(* IEC 61131-3 sources: plc_simulator/services/codesys/POUs (part 6) *)

(* ---- TSK_NoTreatment.st ---- *)
(* ===========================================================================================
 *  TSK_NoTreatment — Create no-treatment transfer tasks
 *
 *  Company : Galvatek part of the John Cockerill Group
 *  Author  : Jarmo Piipponen
 *  Created : 25.03.2026
 *
 * -------------------------------------------------------------------------------------------
 *  Scans units with a target and creates transfer tasks
 *  using the g_ntt destination table.
 *
 *  VAR_IN_OUT: io_task — only mutable array (inserts NTT tasks).
 *  All other globals are read-only via VAR_EXTERNAL.
 *
 *  ------------------------------------------------------------------------------------------
 *
 *  Changes:
 *
 *
 *
 *)

FUNCTION TSK_NoTreatment : BOOL

(* Introduction of Variables ----------------------------------------------------------------*)

VAR_INPUT
  i_time_s                  : LINT;
END_VAR

VAR_IN_OUT  (* array sizes must match GVL_JC_Constants: 3=MAX_TRANSPORTERS *)
  io_task                   : ARRAY[1..3] OF UDT_JC_TskQueueType;
END_VAR

VAR_EXTERNAL CONSTANT
    MAX_TRANSPORTERS        : INT;
    MAX_STATIONS_PER_STEP   : INT;
    MIN_STATION_INDEX        : INT;
    MAX_STATION_INDEX        : INT;
    MAX_UNITS               : INT;
    MAX_TASK_QUEUE          : INT;
    SCH_DISPATCH_MARGIN_S   : REAL;
    NOT_PROCESSED           : INT;
    PROCESSED               : INT;
    USED                    : INT;
END_VAR

VAR_EXTERNAL
  g_unit                    : ARRAY[1..MAX_UNITS] OF UDT_JC_UnitType;
  g_batch                   : ARRAY[1..MAX_UNITS] OF UDT_BatchType;
  g_ntt                     : ARRAY[1..MAX_TRANSPORTERS] OF UDT_JC_NttTransporterType;
  g_transporter             : ARRAY[1..MAX_TRANSPORTERS] OF UDT_TransporterStatusType;
  Stations                 : ARRAY[MIN_STATION_INDEX..MAX_STATION_INDEX] OF UDT_StationType;
  g_station_occupancy             : ARRAY[1..MAX_STATION_INDEX] OF UDT_JC_UnitAtStationType;
  Transporters                     : ARRAY[0..MAX_TRANSPORTERS] OF UDT_TransporterType;
  g_move                    : ARRAY[1..MAX_TRANSPORTERS] OF UDT_JC_MoveTimesType;
END_VAR

VAR
  ui                        : INT;
  loc                       : INT;
  tgt                       : INT;
  cov_t                     : INT;
  ai                        : INT;
  covers                    : BOOL;
  done                      : BOOL;
  dest                      : UDT_JC_NttDestType;
  ntt_idx                   : INT;
  on_primary                : BOOL;
  on_fallback               : BOOL;
  primary_free              : BOOL;
  dest_stn                  : INT;
  si                        : INT;
  station_idx               : INT;
  stn_free                  : BOOL;
  uj                        : INT;
  ti                        : INT;
  already                   : BOOL;
  qi2                       : INT;
  xfer_s                    : REAL;
  task_start                : LINT;
  task_end                  : LINT;
  slot_start                : LINT;
  tmp_move                  : UDT_JC_MoveTimesType;
  slot_end                  : LINT;
  latest_end                : LINT;
  travel_from_sink          : REAL;
  travel_to_lift_s          : REAL;
  trans_pos                 : INT;
  ntt_duration              : LINT;
  slot_ok                   : BOOL;
  sh                        : INT;

  (* Idle-stretch: extend blocking batch CalTime to make room for NTT -----------------------*)
  stretch_pending           : BOOL;
  stretch_unit_id           : INT;
  stretch_deficit           : DINT;
  stretch_avail             : DINT;

  (* Multi-transporter shared-area idle check -----------------------------------------------*)
  ot                        : INT;
  oq                        : INT;
  overlap_conflict          : BOOL;
  dest_x                    : DINT;
  avoid_dist                : DINT;
  cov_min_x                 : DINT;
  cov_max_x                 : DINT;
  ot_min_x                  : DINT;
  ot_max_x                  : DINT;
  zone_min_x                : DINT;
  zone_max_x                : DINT;
  danger_min                : DINT;
  danger_max                : DINT;
  (* Shared-area timing: NTT split into own-area + shared-area portions ---------------------*)
  loc_idx                   : INT;
  loc_x                     : DINT;
  phase2_s                  : REAL;
  shared_entry              : LINT;
  shared_time               : REAL;
  ot_idle_ok                : BOOL;
  ot_idle_start             : LINT;
  ot_idle_end               : LINT;
  ot_next_lift              : INT;
  ot_dispatch_from          : INT;
  ot_travel_to_next         : REAL;

  (* Idle-stretch for other transporter: widen idle gap by extending blocker CalTime --------*)
  ot_stretch_pending        : BOOL;
  ot_stretch_unit_id        : INT;
  ot_stretch_deficit        : DINT;
  ot_stretch_avail          : DINT;
  ot_stretch_need           : LINT;
  ot_stretch_ok             : BOOL;
END_VAR

TSK_NoTreatment := TRUE;

FOR ui := 1 TO MAX_UNITS DO
  tgt := g_unit[ui].Target;
  loc := g_unit[ui].location;

  IF tgt >= 1 AND tgt <= 5 AND loc >= MIN_STATION_INDEX THEN

    IF tgt = 3 AND (g_batch[ui].BatchCode = 0 OR g_batch[ui].State <> NOT_PROCESSED) THEN
      CONTINUE;
    END_IF;

    already := FALSE;
    FOR ti := 1 TO MAX_TRANSPORTERS DO
      IF NOT already THEN
        IF g_transporter[ti].Phase > 0 AND g_station_occupancy[ti].UnitId = ui THEN
          already := TRUE;
        END_IF;
        FOR qi2 := 1 TO io_task[ti].Count DO
          IF NOT already THEN
            IF io_task[ti].Queue[qi2].Unit = ui THEN
              already := TRUE;
            END_IF;
          END_IF;
        END_FOR;
      END_IF;
    END_FOR;

    IF NOT already THEN

    done := FALSE;
    FOR cov_t := 1 TO MAX_TRANSPORTERS DO
      IF NOT done THEN

      covers := FALSE;
      FOR ai := 1 TO 4 DO
        IF NOT covers THEN
          IF Transporters[cov_t].TaskArea[ai].MinLift > 0 OR Transporters[cov_t].TaskArea[ai].MaxLift > 0 THEN
            IF loc >= Transporters[cov_t].TaskArea[ai].MinLift AND loc <= Transporters[cov_t].TaskArea[ai].MaxLift THEN
              covers := TRUE;
            END_IF;
          END_IF;
        END_IF;
      END_FOR;

      IF covers AND g_transporter[cov_t].IsActive
         AND (g_transporter[cov_t].Phase = 0 OR tgt = 5) THEN

        IF tgt = 2 THEN
          IF g_batch[ui].BatchCode = 0 THEN ntt_idx := 6;
          ELSIF g_batch[ui].State = PROCESSED THEN ntt_idx := 8;
  ELSE ntt_idx := 7; END_IF;
        ELSIF tgt = 3 THEN ntt_idx := 7;
  ELSE ntt_idx := tgt; END_IF;

        dest := g_ntt[cov_t].Target[ntt_idx];

        on_primary := FALSE;
        FOR si := 1 TO dest.StationCount DO
  IF dest.Stations[si] = loc THEN on_primary := TRUE; END_IF;
        END_FOR;

        IF NOT on_primary THEN

          on_fallback := FALSE;
          FOR si := 1 TO dest.FallbackCount DO
  IF dest.FallbackStations[si] = loc THEN on_fallback := TRUE; END_IF;
          END_FOR;

          primary_free := FALSE;
          FOR si := 1 TO dest.StationCount DO
            station_idx := dest.Stations[si];
            IF station_idx <> loc AND station_idx >= MIN_STATION_INDEX AND station_idx <= MAX_STATION_INDEX THEN
              stn_free := TRUE;
              FOR uj := 1 TO MAX_UNITS DO
  IF g_unit[uj].location = station_idx AND g_unit[uj].Status = USED THEN stn_free := FALSE; END_IF;
              END_FOR;
  IF stn_free THEN primary_free := TRUE; END_IF;
            END_IF;
          END_FOR;

          dest_stn := 0;

          IF on_fallback AND NOT primary_free THEN
            dest_stn := 0;
          ELSIF on_fallback AND primary_free THEN
            FOR si := 1 TO dest.StationCount DO
              IF dest_stn = 0 THEN
                station_idx := dest.Stations[si];
                IF station_idx <> loc AND station_idx >= MIN_STATION_INDEX AND station_idx <= MAX_STATION_INDEX THEN
                  stn_free := TRUE;
                  FOR uj := 1 TO MAX_UNITS DO
  IF g_unit[uj].location = station_idx AND g_unit[uj].Status = USED THEN stn_free := FALSE; END_IF;
                  END_FOR;
  IF stn_free THEN dest_stn := station_idx; END_IF;
                END_IF;
              END_IF;
            END_FOR;
          ELSE
            FOR si := 1 TO dest.StationCount DO
              IF dest_stn = 0 THEN
                station_idx := dest.Stations[si];
                IF station_idx <> loc AND station_idx >= MIN_STATION_INDEX AND station_idx <= MAX_STATION_INDEX THEN
                  stn_free := TRUE;
                  FOR uj := 1 TO MAX_UNITS DO
  IF g_unit[uj].location = station_idx AND g_unit[uj].Status = USED THEN stn_free := FALSE; END_IF;
                  END_FOR;
  IF stn_free THEN dest_stn := station_idx; END_IF;
                END_IF;
              END_IF;
            END_FOR;

            IF dest_stn = 0 THEN
              FOR si := 1 TO dest.FallbackCount DO
                IF dest_stn = 0 THEN
                  station_idx := dest.FallbackStations[si];
                  IF station_idx <> loc AND station_idx >= MIN_STATION_INDEX AND station_idx <= MAX_STATION_INDEX THEN
                    stn_free := TRUE;
                    FOR uj := 1 TO MAX_UNITS DO
  IF g_unit[uj].location = station_idx AND g_unit[uj].Status = USED THEN stn_free := FALSE; END_IF;
                    END_FOR;
  IF stn_free THEN dest_stn := station_idx; END_IF;
                  END_IF;
                END_IF;
              END_FOR;
            END_IF;
          END_IF;

          IF dest_stn > 0 THEN
            tmp_move := g_move[cov_t];
            xfer_s := STC_CalcTransferTime(
              i_from_stn            := loc,
              i_to_stn              := dest_stn,
              i_move                := tmp_move,
              i_from_dropping_x10   := Stations[loc].DrippingTime,
              i_to_device_delay_x10 := Stations[dest_stn].DeviceDelay,
              i_drip_tray_delay_x10 := Transporters[cov_t].DripTrayDelay);

            (* ── Travel-to: time for transporter to reach lift station ── *)
            travel_to_lift_s := 0.0;
            IF g_transporter[cov_t].Phase = 0 THEN
              trans_pos := g_transporter[cov_t].CurrentStation;
            ELSE
              trans_pos := g_transporter[cov_t].SinkStationTarget;
            END_IF;
            IF trans_pos > 0 AND trans_pos <> loc THEN
              travel_to_lift_s := STC_CalcHorizontalTravel(
                i_from_stn := trans_pos,
                i_to_stn   := loc,
                i_move     := tmp_move);
            END_IF;

            task_start := i_time_s + REAL_TO_LINT(travel_to_lift_s);
            task_end   := task_start + REAL_TO_LINT(xfer_s);
            ntt_duration := task_end - task_start;

            slot_ok := FALSE;
            stretch_pending := FALSE;
            ot_stretch_pending := FALSE;

            IF io_task[cov_t].Count = 0 THEN
              slot_ok := TRUE;
            ELSE
              IF io_task[cov_t].Queue[1].StartTime > task_start THEN
                slot_start := task_start;
                slot_end   := io_task[cov_t].Queue[1].StartTime;
                travel_from_sink := STC_CalcHorizontalTravel(
                  i_from_stn := dest_stn,
                  i_to_stn   := io_task[cov_t].Queue[1].LiftStationTarget,
                  i_move     := g_move[cov_t]);
                latest_end := slot_end - REAL_TO_LINT(travel_from_sink) - 1;
                IF task_start >= slot_start AND task_end <= latest_end THEN
                  slot_ok := TRUE;
                END_IF;

                (* ── Idle-stretch: NTT slightly too long for idle window ──
                   Check if the blocking batch's treatment CalTime can be
                   extended (up to MaxTime) to widen the idle gap.  Only flag
                   the intent here; the actual g_batch write happens after
                   the multi-transporter overlap check passes. *)
                IF NOT slot_ok AND latest_end > 0 THEN
                  stretch_deficit := LINT_TO_DINT(task_end - latest_end);
                  IF stretch_deficit > 0 THEN
                    stretch_unit_id := io_task[cov_t].Queue[1].Unit;
                    IF stretch_unit_id >= 1 AND stretch_unit_id <= MAX_UNITS THEN
                      stretch_avail := g_batch[stretch_unit_id].MaxTime
                                     - g_batch[stretch_unit_id].CalTime;
                      IF stretch_avail >= stretch_deficit THEN
                        stretch_pending := TRUE;
                        slot_ok := TRUE;
                      END_IF;
                    END_IF;
                  END_IF;
                END_IF;
              END_IF;
            END_IF;

            IF NOT slot_ok THEN
              IF io_task[cov_t].Count > 0
                 AND io_task[cov_t].Queue[1].SinkStationTarget = loc THEN
                slot_ok := TRUE;
              ELSE
                dest_stn := 0;
              END_IF;
            END_IF;
          END_IF;

          (* ── Multi-transporter shared-area idle check ──
             If dest_stn is on the shared drive area between two transporters,
             the other transporter must have an idle window covering the time
             when THIS transporter is physically on the shared area.

             NTT transfer phases:
               Phase 2: lift + drip + tray  (nostin on vielä lift-asemalla)
               Phase 3: horizontal travel   (nostin liikkuu kohti dest)
               Phase 4: lower + tray + dev  (nostin on dest-asemalla)

             If lift station is NOT on shared area:
               shared_entry = task_start + phase2_s  (travel starts)
               shared_time  = xfer_s - phase2_s
             If lift station IS on shared area:
               shared_entry = task_start  (already there)
               shared_time  = xfer_s
          *)
          IF dest_stn > 0 THEN
            overlap_conflict := FALSE;
            dest_x := Stations[dest_stn].XPosition;
            avoid_dist := Transporters[cov_t].AvoidanceWidth;
            cov_min_x := Transporters[cov_t].DrivePosMin;
            cov_max_x := Transporters[cov_t].DrivePosMax;

            FOR ot := 1 TO MAX_TRANSPORTERS DO
              IF ot <> cov_t AND NOT overlap_conflict
                 AND g_transporter[ot].IsActive THEN
                ot_min_x := Transporters[ot].DrivePosMin;
                ot_max_x := Transporters[ot].DrivePosMax;

                IF cov_min_x > ot_min_x THEN zone_min_x := cov_min_x;
  ELSE zone_min_x := ot_min_x; END_IF;
                IF cov_max_x < ot_max_x THEN zone_max_x := cov_max_x;
  ELSE zone_max_x := ot_max_x; END_IF;

                IF zone_min_x >= zone_max_x THEN CONTINUE; END_IF;
                IF dest_x < zone_min_x OR dest_x > zone_max_x THEN CONTINUE; END_IF;

                danger_min := zone_min_x - avoid_dist;
                danger_max := zone_max_x + avoid_dist;

                (* ── Calculate shared-area entry time and duration ── *)
                loc_x := Stations[loc].XPosition;
                IF loc_x >= danger_min AND loc_x <= danger_max THEN
                  shared_entry := task_start;
                  shared_time  := xfer_s;
                ELSE
                  loc_idx := loc - MIN_STATION_INDEX;
                  IF loc_idx >= 1 AND loc_idx <= 25 THEN
                    phase2_s := INT_TO_REAL(g_move[cov_t].LiftTime[loc_idx]) / 10.0
                              + INT_TO_REAL(Stations[loc].DrippingTime) / 10.0
                              + INT_TO_REAL(Transporters[cov_t].DripTrayDelay) / 10.0;
                  ELSE
                    phase2_s := 0.0;
                  END_IF;
                  shared_entry := task_start + REAL_TO_LINT(phase2_s);
                  shared_time  := xfer_s - phase2_s;
  IF shared_time < 1.0 THEN shared_time := 1.0; END_IF;
                END_IF;

                (* ── Check: does other transporter have an idle window
                     that starts ≤ shared_entry and lasts ≥ shared_time? ── *)
                ot_idle_ok := FALSE;

                IF io_task[ot].Count = 0 AND g_transporter[ot].Phase = 0 THEN
                  ot_idle_ok := TRUE;
                ELSIF io_task[ot].Count = 0
                      AND g_transporter[ot].Phase >= 1
                      AND g_transporter[ot].Phase <= 4 THEN
                  (* Transporter executing task, nothing queued after.
                     Idle starts at current task finish. *)
                  ot_idle_start := g_transporter[ot].CurrentTaskFinishTime;
                  IF ot_idle_start <= shared_entry THEN
                    ot_idle_ok := TRUE;
                  END_IF;
                ELSE
                  IF io_task[ot].Count > 0 THEN
                    IF g_transporter[ot].Phase >= 1 AND g_transporter[ot].Phase <= 4 THEN
                      (* Idle gap: current task finish → next queued start *)
                      ot_idle_start := g_transporter[ot].CurrentTaskFinishTime;
                      ot_dispatch_from := g_transporter[ot].SinkStationTarget;
                    ELSE
                      ot_idle_start := task_start;
                      ot_dispatch_from := g_transporter[ot].CurrentStation;
                    END_IF;
                    ot_next_lift := io_task[ot].Queue[1].LiftStationTarget;
                    ot_travel_to_next := 0.0;
                    IF ot_dispatch_from > 0
                       AND ot_next_lift > 0
                       AND ot_dispatch_from <> ot_next_lift THEN
                      ot_travel_to_next := STC_CalcHorizontalTravel(
                        i_from_stn := ot_dispatch_from,
                        i_to_stn   := ot_next_lift,
                        i_move     := g_move[ot]);
                    END_IF;
                    ot_idle_end := io_task[ot].Queue[1].StartTime
                                 - REAL_TO_LINT(ot_travel_to_next)
                                 - REAL_TO_LINT(SCH_DISPATCH_MARGIN_S);
                    IF ot_idle_end < ot_idle_start THEN
                      ot_idle_end := ot_idle_start;
                    END_IF;
                    IF ot_idle_start <= shared_entry
                       AND ot_idle_end >= shared_entry + REAL_TO_LINT(shared_time) THEN
                      ot_idle_ok := TRUE;
                    END_IF;
                  END_IF;

                  IF NOT ot_idle_ok THEN
                    FOR oq := 1 TO io_task[ot].Count - 1 DO
                      IF NOT ot_idle_ok THEN
                        ot_idle_start := io_task[ot].Queue[oq].FinishTime;
                        ot_dispatch_from := io_task[ot].Queue[oq].SinkStationTarget;
                        ot_next_lift := io_task[ot].Queue[oq + 1].LiftStationTarget;
                        ot_travel_to_next := 0.0;
                        IF ot_dispatch_from > 0
                           AND ot_next_lift > 0
                           AND ot_dispatch_from <> ot_next_lift THEN
                          ot_travel_to_next := STC_CalcHorizontalTravel(
                            i_from_stn := ot_dispatch_from,
                            i_to_stn   := ot_next_lift,
                            i_move     := g_move[ot]);
                        END_IF;
                        ot_idle_end := io_task[ot].Queue[oq + 1].StartTime
                                     - REAL_TO_LINT(ot_travel_to_next)
                                     - REAL_TO_LINT(SCH_DISPATCH_MARGIN_S);
                        IF ot_idle_end < ot_idle_start THEN
                          ot_idle_end := ot_idle_start;
                        END_IF;
                        IF ot_idle_start <= shared_entry
                           AND ot_idle_end >= shared_entry + REAL_TO_LINT(shared_time) THEN
                          ot_idle_ok := TRUE;
                        END_IF;
                      END_IF;
                    END_FOR;
                  END_IF;

                  IF NOT ot_idle_ok AND io_task[ot].Count > 0 THEN
                    ot_idle_start := io_task[ot].Queue[io_task[ot].Count].FinishTime;
                    IF ot_idle_start <= shared_entry THEN
                      ot_idle_ok := TRUE;
                    END_IF;
                  END_IF;
                END_IF;

                IF NOT ot_idle_ok THEN
                  (* ── Idle-stretch for other transporter ──
                     Try to widen the nearest idle gap by extending the
                     blocking batch CalTime (up to MaxTime).  Only tasks
                     with Stage > 0 (regular, not NTT) are candidates. *)
                  ot_stretch_ok := FALSE;

                  (* Try gap before first task *)
                  IF io_task[ot].Count > 0
                     AND io_task[ot].Queue[1].Stage > 0 THEN
                    IF g_transporter[ot].Phase >= 1 AND g_transporter[ot].Phase <= 4 THEN
                      ot_idle_start := g_transporter[ot].CurrentTaskFinishTime;
                      ot_dispatch_from := g_transporter[ot].SinkStationTarget;
                    ELSE
                      ot_idle_start := task_start;
                      ot_dispatch_from := g_transporter[ot].CurrentStation;
                    END_IF;
                    ot_next_lift := io_task[ot].Queue[1].LiftStationTarget;
                    ot_travel_to_next := 0.0;
                    IF ot_dispatch_from > 0
                       AND ot_next_lift > 0
                       AND ot_dispatch_from <> ot_next_lift THEN
                      ot_travel_to_next := STC_CalcHorizontalTravel(
                        i_from_stn := ot_dispatch_from,
                        i_to_stn   := ot_next_lift,
                        i_move     := g_move[ot]);
                    END_IF;
                    ot_idle_end := io_task[ot].Queue[1].StartTime
                                 - REAL_TO_LINT(ot_travel_to_next)
                                 - REAL_TO_LINT(SCH_DISPATCH_MARGIN_S);
                    IF ot_idle_end < ot_idle_start THEN
                      ot_idle_end := ot_idle_start;
                    END_IF;

                    IF ot_idle_start <= shared_entry
                       AND ot_idle_end > shared_entry THEN
                      ot_stretch_need := shared_entry
                                       + REAL_TO_LINT(shared_time)
                                       - ot_idle_end;
                      IF ot_stretch_need > LINT#0 THEN
                        ot_stretch_unit_id := io_task[ot].Queue[1].Unit;
                        IF ot_stretch_unit_id >= 1
                           AND ot_stretch_unit_id <= MAX_UNITS THEN
                          ot_stretch_avail :=
                            g_batch[ot_stretch_unit_id].MaxTime
                          - g_batch[ot_stretch_unit_id].CalTime;
                          IF ot_stretch_avail >= LINT_TO_DINT(ot_stretch_need) THEN
                            ot_stretch_deficit := LINT_TO_DINT(ot_stretch_need);
                            ot_stretch_pending := TRUE;
                            ot_stretch_ok      := TRUE;
                          END_IF;
                        END_IF;
                      END_IF;
                    END_IF;
                  END_IF;

                  (* Try gaps between tasks *)
                  IF NOT ot_stretch_ok THEN
                    FOR oq := 1 TO io_task[ot].Count - 1 DO
                      IF NOT ot_stretch_ok
                         AND io_task[ot].Queue[oq + 1].Stage > 0 THEN
                        ot_idle_start := io_task[ot].Queue[oq].FinishTime;
                        ot_dispatch_from := io_task[ot].Queue[oq].SinkStationTarget;
                        ot_next_lift := io_task[ot].Queue[oq + 1].LiftStationTarget;
                        ot_travel_to_next := 0.0;
                        IF ot_dispatch_from > 0
                           AND ot_next_lift > 0
                           AND ot_dispatch_from <> ot_next_lift THEN
                          ot_travel_to_next := STC_CalcHorizontalTravel(
                            i_from_stn := ot_dispatch_from,
                            i_to_stn   := ot_next_lift,
                            i_move     := g_move[ot]);
                        END_IF;
                        ot_idle_end := io_task[ot].Queue[oq + 1].StartTime
                                     - REAL_TO_LINT(ot_travel_to_next)
                                     - REAL_TO_LINT(SCH_DISPATCH_MARGIN_S);
                        IF ot_idle_end < ot_idle_start THEN
                          ot_idle_end := ot_idle_start;
                        END_IF;

                        IF ot_idle_start <= shared_entry
                           AND ot_idle_end > shared_entry THEN
                          ot_stretch_need := shared_entry
                                           + REAL_TO_LINT(shared_time)
                                           - ot_idle_end;
                          IF ot_stretch_need > LINT#0 THEN
                            ot_stretch_unit_id := io_task[ot].Queue[oq + 1].Unit;
                            IF ot_stretch_unit_id >= 1
                               AND ot_stretch_unit_id <= MAX_UNITS THEN
                              ot_stretch_avail :=
                                g_batch[ot_stretch_unit_id].MaxTime
                              - g_batch[ot_stretch_unit_id].CalTime;
                              IF ot_stretch_avail >= LINT_TO_DINT(ot_stretch_need) THEN
                                ot_stretch_deficit := LINT_TO_DINT(ot_stretch_need);
                                ot_stretch_pending := TRUE;
                                ot_stretch_ok      := TRUE;
                              END_IF;
                            END_IF;
                          END_IF;
                        END_IF;
                      END_IF;
                    END_FOR;
                  END_IF;

                  IF ot_stretch_ok THEN
                    ot_idle_ok := TRUE;
                  ELSE
                    overlap_conflict := TRUE;
                  END_IF;
                END_IF;
              END_IF;
            END_FOR;

  IF overlap_conflict THEN dest_stn := 0; END_IF;
          END_IF;

          IF dest_stn > 0 THEN
            (* ── Commit idle-stretch: extend blocking batch CalTime ── *)
            IF stretch_pending THEN
              g_batch[stretch_unit_id].CalTime :=
                g_batch[stretch_unit_id].CalTime + stretch_deficit;
              stretch_pending := FALSE;
            END_IF;

            (* ── Commit other-transporter idle-stretch ── *)
            IF ot_stretch_pending THEN
              g_batch[ot_stretch_unit_id].CalTime :=
                g_batch[ot_stretch_unit_id].CalTime + ot_stretch_deficit;
              ot_stretch_pending := FALSE;
            END_IF;

            IF io_task[cov_t].Count < MAX_TASK_QUEUE THEN
              FOR sh := io_task[cov_t].Count TO 1 BY -1 DO
                io_task[cov_t].Queue[sh + 1] := io_task[cov_t].Queue[sh];
              END_FOR;
              io_task[cov_t].Queue[1].Unit         := ui;
              io_task[cov_t].Queue[1].Stage        := 0;
              io_task[cov_t].Queue[1].LiftStationTarget := loc;
              io_task[cov_t].Queue[1].SinkStationTarget := dest_stn;
              io_task[cov_t].Queue[1].StartTime   := task_start;
              io_task[cov_t].Queue[1].FinishTime  := task_end;
              io_task[cov_t].Queue[1].CalcTime    := 0;
              io_task[cov_t].Queue[1].MinTime     := 0;
              io_task[cov_t].Queue[1].MaxTime     := 0;
              io_task[cov_t].Queue[1].NttPrimary := 0;
              FOR si := 1 TO dest.StationCount DO
                IF dest.Stations[si] = dest_stn THEN
                  io_task[cov_t].Queue[1].NttPrimary := 1;
                END_IF;
              END_FOR;
              io_task[cov_t].Count := io_task[cov_t].Count + 1;
              done := TRUE;
            END_IF;
          END_IF;

        END_IF; (* NOT on_primary *)
      END_IF; (* covers + idle *)
      END_IF; (* NOT done *)
    END_FOR; (* transporter loop *)
    END_IF; (* NOT already *)
  END_IF; (* valid target *)
END_FOR;

END_FUNCTION

(* ---- TSK_Resolve.st ---- *)
(* ===========================================================================================
 *  TSK_Resolve — Conflict resolution
 *
 *  Company : Galvatek part of the John Cockerill Group
 *  Author  : Jarmo Piipponen
 *  Created : 25.03.2026
 *
 * -------------------------------------------------------------------------------------------
 *  Four sequential resolution phases:
 *  1. ADVANCE (chain bottleneck + suffix flex_down)
 *  2. DELAY (single-stage flex_up)
 *  3. PRECEDING_DELAY (conf stage-1)
 *  4. DELAY_PREV_PAST_NEXT (force order swap)
 *
 *  VAR_IN_OUT: io_schedule, io_task, io_batch, io_locks,
 *  io_lock_cnt — caller passes live or workspace arrays.
 *
 *  ------------------------------------------------------------------------------------------
 *
 *  Changes:
 *
 *
 *
 *)

FUNCTION TSK_Resolve : BOOL

(* Introduction of Variables ----------------------------------------------------------------*)

VAR_INPUT
  i_conf_unit               : INT;
  i_conf_stage              : INT;
  i_conf_trans              : INT;
  i_blocked_unit            : INT;
  i_blocked_stage           : INT;
  i_deficit                 : REAL;
END_VAR

VAR_IN_OUT  (* array sizes must match GVL_JC_Constants: 50=MAX_LOCKS, 10=MAX_UNITS, 3=MAX_TRANSPORTERS *)
  io_locks                  : ARRAY[1..50] OF UDT_JC_TskLockType;
  io_lock_cnt               : INT;
  io_schedule               : ARRAY[1..10] OF UDT_JC_TskScheduleType;
  io_task                   : ARRAY[1..3] OF UDT_JC_TskQueueType;
  io_batch                  : ARRAY[1..10] OF UDT_BatchType;
END_VAR

VAR_EXTERNAL CONSTANT
    MAX_TRANSPORTERS        : INT;
    MAX_UNITS               : INT;
    SCH_TSK_FLEX_FACTOR     : REAL;
END_VAR

VAR_OUTPUT
  o_solved                  : BOOL;
  o_total_delay             : REAL;
  o_total_adv               : REAL;
END_VAR

VAR
  remain                    : REAL;
  cap                       : REAL;
  amount                    : REAL;
  stage_flex                : REAL;
  is_locked_adv             : BOOL;
  is_locked_del             : BOOL;
  can_advance               : BOOL;
  can_delay                 : BOOL;
  lock_i                    : INT;
  prev_conf_stage           : INT;
  is_pcs_locked             : BOOL;
  prev_sink_stn             : INT;
  next_lift_stn             : INT;
  is_blk_adv_locked         : BOOL;
  qi                        : INT;
  chain_flex                : REAL;
  suffix_flex               : REAL;
  earlier_stg               : INT;
  earlier_flex              : REAL;
  chain_amount              : REAL;
  suffix_amount             : REAL;
  sched_blocked             : INT;
  sched_conf                : INT;
  sched_prev_conf           : INT;
  tmp_si                    : INT;
  cap_remain                : REAL;
END_VAR

TSK_Resolve := FALSE;
o_solved      := FALSE;
o_total_delay := 0.0;
o_total_adv   := 0.0;
remain        := i_deficit;

IF remain <= 0.1 THEN
  o_solved := TRUE;
  TSK_Resolve := TRUE;
  RETURN;
END_IF;

(* Lock check: blocked stage locked DELAY? cannot ADVANCE *)
is_locked_adv := FALSE;
FOR lock_i := 1 TO io_lock_cnt DO
  IF io_locks[lock_i].Unit = i_blocked_unit
     AND io_locks[lock_i].Stage = i_blocked_stage
     AND io_locks[lock_i].Direction = 2 THEN
    is_locked_adv := TRUE;
  END_IF;
END_FOR;

(* Lock check: conf stage locked ADVANCE? cannot DELAY *)
is_locked_del := FALSE;
FOR lock_i := 1 TO io_lock_cnt DO
  IF io_locks[lock_i].Unit = i_conf_unit
     AND io_locks[lock_i].Stage = i_conf_stage
     AND io_locks[lock_i].Direction = 1 THEN
    is_locked_del := TRUE;
  END_IF;
END_FOR;

can_advance := NOT is_locked_adv;
can_delay   := NOT is_locked_del;

(* Map ProgramStage to schedule array index *)
sched_blocked := 0;
IF i_blocked_unit >= 1 AND i_blocked_unit <= MAX_UNITS THEN
  FOR tmp_si := 1 TO io_schedule[i_blocked_unit].StageCount DO
    IF io_schedule[i_blocked_unit].Stages[tmp_si].ProgramStage = i_blocked_stage THEN
      sched_blocked := tmp_si; EXIT;
    END_IF;
  END_FOR;
END_IF;

sched_conf := 0;
IF i_conf_unit >= 1 AND i_conf_unit <= MAX_UNITS THEN
  FOR tmp_si := 1 TO io_schedule[i_conf_unit].StageCount DO
    IF io_schedule[i_conf_unit].Stages[tmp_si].ProgramStage = i_conf_stage THEN
      sched_conf := tmp_si; EXIT;
    END_IF;
  END_FOR;
END_IF;

(* ================================================================ *)
(* PHASE 1: ADVANCE -- advance blocked batch                       *)
(* ================================================================ *)
IF can_advance
   AND i_blocked_unit >= 1 AND i_blocked_unit <= MAX_UNITS
   AND i_blocked_stage >= 1 THEN
IF sched_blocked >= 1 AND sched_blocked <= io_schedule[i_blocked_unit].StageCount THEN

  (* Absolute flex cap: use (MaxTime - MinTime) range, not (CalcTime - MinTime).
     This prevents cumulative drift when CalcTime is adjusted across rounds. *)
  stage_flex := DINT_TO_REAL(
    io_schedule[i_blocked_unit].Stages[sched_blocked].MaxTime
    - io_schedule[i_blocked_unit].Stages[sched_blocked].MinTime);
  IF stage_flex < 0.0 THEN stage_flex := 0.0; END_IF;
  stage_flex := stage_flex * SCH_TSK_FLEX_FACTOR;
  (* Cap to actual remaining advance room *)
  cap_remain := DINT_TO_REAL(
    io_schedule[i_blocked_unit].Stages[sched_blocked].CalcTime
    - io_schedule[i_blocked_unit].Stages[sched_blocked].MinTime);
  IF cap_remain < 0.0 THEN cap_remain := 0.0; END_IF;
  IF stage_flex > cap_remain THEN stage_flex := cap_remain; END_IF;

  IF stage_flex > 0.1 THEN
    IF io_batch[i_blocked_unit].CurStage = i_blocked_stage THEN cap := 0.9;
  ELSE cap := 0.5; END_IF;

    (* Chain bottleneck search *)
    chain_flex := stage_flex;
    FOR earlier_stg := 1 TO sched_blocked - 1 DO
      earlier_flex := DINT_TO_REAL(
        io_schedule[i_blocked_unit].Stages[earlier_stg].CalcTime
        - io_schedule[i_blocked_unit].Stages[earlier_stg].MinTime);
  IF earlier_flex < 0.0 THEN earlier_flex := 0.0; END_IF;
      IF earlier_flex > 0.0 AND earlier_flex < chain_flex THEN
        chain_flex := earlier_flex;
      END_IF;
    END_FOR;

    (* CHAIN_ADVANCE *)
    chain_amount := chain_flex * cap;
  IF chain_amount > remain THEN chain_amount := remain; END_IF;

    IF chain_amount > 0.1 THEN
      io_schedule[i_blocked_unit].Stages[sched_blocked].CalcTime :=
        io_schedule[i_blocked_unit].Stages[sched_blocked].CalcTime - REAL_TO_DINT(chain_amount);
      io_schedule[i_blocked_unit].Stages[sched_blocked].ExitTime :=
        io_schedule[i_blocked_unit].Stages[sched_blocked].ExitTime - REAL_TO_LINT(chain_amount);

      STC_ShiftSchedule(i_unit := i_blocked_unit, i_from_stage := i_blocked_stage + 1,
                         i_amount := -chain_amount, io_schedule := io_schedule, io_task := io_task);

      io_batch[i_blocked_unit].CalTime :=
        io_batch[i_blocked_unit].CalTime - REAL_TO_DINT(chain_amount);
      IF io_batch[i_blocked_unit].CalTime < io_batch[i_blocked_unit].MinTime THEN
        io_batch[i_blocked_unit].CalTime := io_batch[i_blocked_unit].MinTime;
      END_IF;

      remain := remain - chain_amount;
      o_total_adv := o_total_adv + chain_amount;
    END_IF;

    (* SUFFIX_ADVANCE *)
    suffix_flex := stage_flex - chain_flex;
    IF suffix_flex > 0.1 AND remain > 0.1 THEN
      suffix_amount := suffix_flex * cap;
  IF suffix_amount > remain THEN suffix_amount := remain; END_IF;

      IF suffix_amount > 0.1 THEN
        io_schedule[i_blocked_unit].Stages[sched_blocked].CalcTime :=
          io_schedule[i_blocked_unit].Stages[sched_blocked].CalcTime - REAL_TO_DINT(suffix_amount);
        io_schedule[i_blocked_unit].Stages[sched_blocked].ExitTime :=
          io_schedule[i_blocked_unit].Stages[sched_blocked].ExitTime - REAL_TO_LINT(suffix_amount);

        STC_ShiftSchedule(i_unit := i_blocked_unit, i_from_stage := i_blocked_stage + 1,
                           i_amount := -suffix_amount, io_schedule := io_schedule, io_task := io_task);

        io_batch[i_blocked_unit].CalTime :=
          io_batch[i_blocked_unit].CalTime - REAL_TO_DINT(suffix_amount);
        IF io_batch[i_blocked_unit].CalTime < io_batch[i_blocked_unit].MinTime THEN
          io_batch[i_blocked_unit].CalTime := io_batch[i_blocked_unit].MinTime;
        END_IF;

        remain := remain - suffix_amount;
        o_total_adv := o_total_adv + suffix_amount;
      END_IF;
    END_IF;

    (* Record lock: ADVANCE on blocked stage *)
    IF io_lock_cnt < 50 THEN
      io_lock_cnt := io_lock_cnt + 1;
      io_locks[io_lock_cnt].Unit := i_blocked_unit;
      io_locks[io_lock_cnt].Stage := i_blocked_stage;
      io_locks[io_lock_cnt].Direction := 1;
    END_IF;

    IF remain <= 0.1 THEN
  o_solved := TRUE;
  TSK_Resolve := TRUE; RETURN;
    END_IF;
  END_IF;
END_IF;
END_IF;

(* ================================================================ *)
(* PHASE 2: DELAY -- delay conflict batch                          *)
(* ================================================================ *)
IF can_delay AND remain > 0.1
   AND i_conf_unit >= 1 AND i_conf_unit <= MAX_UNITS
   AND i_conf_stage >= 1 THEN
IF sched_conf >= 1 AND sched_conf <= io_schedule[i_conf_unit].StageCount THEN

  (* Absolute flex cap: use (MaxTime - MinTime) range, not (MaxTime - CalcTime).
     This prevents cumulative drift when CalcTime is adjusted across rounds. *)
  stage_flex := DINT_TO_REAL(
    io_schedule[i_conf_unit].Stages[sched_conf].MaxTime
    - io_schedule[i_conf_unit].Stages[sched_conf].MinTime);
  IF stage_flex < 0.0 THEN stage_flex := 0.0; END_IF;
  stage_flex := stage_flex * SCH_TSK_FLEX_FACTOR;
  (* Cap to actual remaining delay room *)
  cap_remain := DINT_TO_REAL(
    io_schedule[i_conf_unit].Stages[sched_conf].MaxTime
    - io_schedule[i_conf_unit].Stages[sched_conf].CalcTime);
  IF cap_remain < 0.0 THEN cap_remain := 0.0; END_IF;
  IF stage_flex > cap_remain THEN stage_flex := cap_remain; END_IF;

  IF stage_flex > 0.1 THEN
    IF io_batch[i_conf_unit].CurStage = i_conf_stage THEN cap := 0.9;
  ELSE cap := 0.5; END_IF;
    amount := stage_flex * cap;
  IF amount > remain THEN amount := remain; END_IF;

    io_schedule[i_conf_unit].Stages[sched_conf].CalcTime :=
      io_schedule[i_conf_unit].Stages[sched_conf].CalcTime + REAL_TO_DINT(amount);
    io_schedule[i_conf_unit].Stages[sched_conf].ExitTime :=
      io_schedule[i_conf_unit].Stages[sched_conf].ExitTime + REAL_TO_LINT(amount);

    STC_ShiftSchedule(i_unit := i_conf_unit, i_from_stage := i_conf_stage + 1,
                       i_amount := amount, io_schedule := io_schedule, io_task := io_task);

    IF io_batch[i_conf_unit].CurStage = i_conf_stage THEN
      io_batch[i_conf_unit].CalTime :=
        io_batch[i_conf_unit].CalTime + REAL_TO_DINT(amount);
      IF io_batch[i_conf_unit].CalTime > io_batch[i_conf_unit].MaxTime THEN
        io_batch[i_conf_unit].CalTime := io_batch[i_conf_unit].MaxTime;
      END_IF;
    END_IF;

    remain := remain - amount;
    o_total_delay := o_total_delay + amount;

    IF io_lock_cnt < 50 THEN
      io_lock_cnt := io_lock_cnt + 1;
      io_locks[io_lock_cnt].Unit := i_conf_unit;
      io_locks[io_lock_cnt].Stage := i_conf_stage;
      io_locks[io_lock_cnt].Direction := 2;
    END_IF;

    IF remain <= 0.1 THEN
  o_solved := TRUE;
  TSK_Resolve := TRUE; RETURN;
    END_IF;
  END_IF;
END_IF;
END_IF;

(* ================================================================ *)
(* PHASE 3: PRECEDING_DELAY -- delay conf batch at stage-1         *)
(* ================================================================ *)
prev_conf_stage := i_conf_stage - 1;

sched_prev_conf := 0;
IF i_conf_unit >= 1 AND i_conf_unit <= MAX_UNITS AND prev_conf_stage >= 1 THEN
  FOR tmp_si := 1 TO io_schedule[i_conf_unit].StageCount DO
    IF io_schedule[i_conf_unit].Stages[tmp_si].ProgramStage = prev_conf_stage THEN
  sched_prev_conf := tmp_si; EXIT;
    END_IF;
  END_FOR;
END_IF;

IF remain > 0.1 AND prev_conf_stage >= 1 AND i_conf_unit >= 1 AND i_conf_unit <= MAX_UNITS
   AND sched_prev_conf >= 1 THEN
  is_pcs_locked := FALSE;
  FOR lock_i := 1 TO io_lock_cnt DO
    IF io_locks[lock_i].Unit = i_conf_unit
       AND io_locks[lock_i].Stage = prev_conf_stage
       AND io_locks[lock_i].Direction = 1 THEN
      is_pcs_locked := TRUE;
    END_IF;
  END_FOR;

  IF NOT is_pcs_locked THEN
    (* Flex cap: min + factor × (max - min); available room = flex_cap - CalcTime *)
    stage_flex := DINT_TO_REAL(
      io_schedule[i_conf_unit].Stages[sched_prev_conf].MinTime
      + REAL_TO_DINT(SCH_TSK_FLEX_FACTOR * DINT_TO_REAL(
          io_schedule[i_conf_unit].Stages[sched_prev_conf].MaxTime
        - io_schedule[i_conf_unit].Stages[sched_prev_conf].MinTime))
      - io_schedule[i_conf_unit].Stages[sched_prev_conf].CalcTime);
  IF stage_flex < 0.0 THEN stage_flex := 0.0; END_IF;

    IF stage_flex > 0.1 THEN
      IF io_batch[i_conf_unit].CurStage = prev_conf_stage THEN cap := 0.9;
  ELSE cap := 0.5; END_IF;
      amount := stage_flex * cap;
  IF amount > remain THEN amount := remain; END_IF;

      io_schedule[i_conf_unit].Stages[sched_prev_conf].CalcTime :=
        io_schedule[i_conf_unit].Stages[sched_prev_conf].CalcTime + REAL_TO_DINT(amount);
      io_schedule[i_conf_unit].Stages[sched_prev_conf].ExitTime :=
        io_schedule[i_conf_unit].Stages[sched_prev_conf].ExitTime + REAL_TO_LINT(amount);
      STC_ShiftSchedule(i_unit := i_conf_unit, i_from_stage := prev_conf_stage + 1,
                         i_amount := amount, io_schedule := io_schedule, io_task := io_task);

      IF io_batch[i_conf_unit].CurStage = i_conf_stage THEN
        io_batch[i_conf_unit].CalTime :=
          io_batch[i_conf_unit].CalTime + REAL_TO_DINT(amount);
        IF io_batch[i_conf_unit].CalTime > io_batch[i_conf_unit].MaxTime THEN
          io_batch[i_conf_unit].CalTime := io_batch[i_conf_unit].MaxTime;
        END_IF;
      END_IF;

      remain := remain - amount;
      o_total_delay := o_total_delay + amount;

      IF io_lock_cnt < 50 THEN
        io_lock_cnt := io_lock_cnt + 1;
        io_locks[io_lock_cnt].Unit := i_conf_unit;
        io_locks[io_lock_cnt].Stage := prev_conf_stage;
        io_locks[io_lock_cnt].Direction := 2;
      END_IF;

      IF remain <= 0.1 THEN
  o_solved := TRUE;
  TSK_Resolve := TRUE; RETURN;
      END_IF;
    END_IF;
  END_IF;
END_IF;

(* ================================================================ *)
(* PHASE 4: DELAY_PREV_PAST_NEXT -- force order swap               *)
(* ================================================================ *)
IF remain > 0.1 AND i_blocked_unit >= 1 AND i_blocked_unit <= MAX_UNITS THEN
  prev_sink_stn := 0;
  next_lift_stn := 0;
  IF i_conf_trans >= 1 AND i_conf_trans <= MAX_TRANSPORTERS THEN
    FOR qi := 1 TO io_task[i_conf_trans].Count DO
      IF io_task[i_conf_trans].Queue[qi].Unit = i_blocked_unit
         AND io_task[i_conf_trans].Queue[qi].Stage = i_blocked_stage THEN
        prev_sink_stn := io_task[i_conf_trans].Queue[qi].SinkStationTarget;
      END_IF;
      IF io_task[i_conf_trans].Queue[qi].Unit = i_conf_unit
         AND io_task[i_conf_trans].Queue[qi].Stage = i_conf_stage THEN
        next_lift_stn := io_task[i_conf_trans].Queue[qi].LiftStationTarget;
      END_IF;
    END_FOR;
  END_IF;

  IF NOT (prev_sink_stn > 0 AND next_lift_stn > 0 AND prev_sink_stn = next_lift_stn) THEN
    is_blk_adv_locked := FALSE;
    FOR lock_i := 1 TO io_lock_cnt DO
      IF io_locks[lock_i].Unit = i_blocked_unit
         AND io_locks[lock_i].Stage = i_blocked_stage
         AND io_locks[lock_i].Direction = 1 THEN
        is_blk_adv_locked := TRUE;
      END_IF;
    END_FOR;

    IF NOT is_blk_adv_locked THEN
      (* Flex cap: min + factor × (max - min); available room = flex_cap - CalcTime *)
      stage_flex := DINT_TO_REAL(
        io_schedule[i_blocked_unit].Stages[sched_blocked].MinTime
        + REAL_TO_DINT(SCH_TSK_FLEX_FACTOR * DINT_TO_REAL(
            io_schedule[i_blocked_unit].Stages[sched_blocked].MaxTime
          - io_schedule[i_blocked_unit].Stages[sched_blocked].MinTime))
        - io_schedule[i_blocked_unit].Stages[sched_blocked].CalcTime);
  IF stage_flex < 0.0 THEN stage_flex := 0.0; END_IF;

      IF stage_flex > 0.1 THEN
        IF io_batch[i_blocked_unit].CurStage = i_blocked_stage THEN cap := 0.9;
  ELSE cap := 0.5; END_IF;
        amount := stage_flex * cap;
  IF amount > remain THEN amount := remain; END_IF;

        io_schedule[i_blocked_unit].Stages[sched_blocked].CalcTime :=
          io_schedule[i_blocked_unit].Stages[sched_blocked].CalcTime + REAL_TO_DINT(amount);
        io_schedule[i_blocked_unit].Stages[sched_blocked].ExitTime :=
          io_schedule[i_blocked_unit].Stages[sched_blocked].ExitTime + REAL_TO_LINT(amount);
        STC_ShiftSchedule(i_unit := i_blocked_unit, i_from_stage := i_blocked_stage + 1,
                           i_amount := amount, io_schedule := io_schedule, io_task := io_task);

        IF io_batch[i_blocked_unit].CurStage = i_blocked_stage THEN
          io_batch[i_blocked_unit].CalTime :=
            io_batch[i_blocked_unit].CalTime + REAL_TO_DINT(amount);
          IF io_batch[i_blocked_unit].CalTime > io_batch[i_blocked_unit].MaxTime THEN
            io_batch[i_blocked_unit].CalTime := io_batch[i_blocked_unit].MaxTime;
          END_IF;
        END_IF;

        remain := remain - amount;
        o_total_delay := o_total_delay + amount;

        IF io_lock_cnt < 50 THEN
          io_lock_cnt := io_lock_cnt + 1;
          io_locks[io_lock_cnt].Unit := i_blocked_unit;
          io_locks[io_lock_cnt].Stage := i_blocked_stage;
          io_locks[io_lock_cnt].Direction := 2;
        END_IF;

        IF remain <= 0.1 THEN
  o_solved := TRUE;
  TSK_Resolve := TRUE; RETURN;
        END_IF;
      END_IF;
    END_IF;
  END_IF;
END_IF;

END_FUNCTION

(* ---- TWA_CalcPriority.st ---- *)
(* ============================================================
   TWA_CalcPriority.st — Priority calculation for collision avoidance

   Priority rules (from transporterWorkingArea.js):
     canEvade = FALSE  → 100000 (cannot move, others must avoid)
     phase 3 (to_sink) → 200000 + (99999 - distance_to_target)
     phase 1 (to_lift) → 100000 + (99999 - distance_to_target)
     phase 0 (idle)    → 1

   Returns REAL to avoid DINT compatibility issues.
   Values fit within REAL precision (max ~300000).
   ============================================================ *)

FUNCTION TWA_CalcPriority : DINT
VAR_INPUT
  i_phase     : INT;
  i_can_evade : BOOL;
  i_x_pos     : DINT;
  i_x_target  : DINT;
END_VAR
VAR
  dist : DINT;
END_VAR

IF NOT i_can_evade THEN
  TWA_CalcPriority := DINT#100000;
  RETURN;
END_IF;

IF i_phase = 3 THEN
  dist := ABS(i_x_pos - i_x_target);
  IF dist > 99999 THEN dist := 99999; END_IF;
  TWA_CalcPriority := DINT#200000 + (DINT#99999 - dist);
ELSIF i_phase = 1 THEN
  dist := ABS(i_x_pos - i_x_target);
  IF dist > 99999 THEN dist := 99999; END_IF;
  TWA_CalcPriority := DINT#100000 + (DINT#99999 - dist);
ELSE
  TWA_CalcPriority := 1;
END_IF;

END_FUNCTION

(* ---- DEP_FB_CalcIdleSlots.st ---- *)
(* ============================================================
   DEP_FB_CalcIdleSlots — Idle slot calculation per transporter
   ============================================================
   Calculates time windows where a transporter has no tasks.
   Each gap between consecutive tasks (or before the first /
   after the last task) is an idle slot.

   Source: transporterTaskScheduler.js calculateTransporterIdleSlots()

   Expects g_task[i_trans].Queue to be already sorted by start_time
   (TSK_FB_Scheduler TASKS_SORT phase ensures this).

   Used by: DEP_FB_Scheduler (CHECK_ANALYZE phase)
   ============================================================ *)

FUNCTION_BLOCK DEP_FB_CalcIdleSlots
VAR_INPUT
  i_trans  : INT;      (* transporter index 1..3 *)
  i_time_s : LINT;     (* current simulation time (s), unix seconds *)
END_VAR
VAR_EXTERNAL CONSTANT
    MAX_Transporters   : INT;
    MAX_Units          : INT;
    DEP_MAX_IDLE_SLOTS : INT;
END_VAR

VAR_EXTERNAL
  g_task          : ARRAY[1..MAX_Transporters] OF UDT_JC_TskQueueType;
  g_dep_idle_slot : ARRAY[1..MAX_Transporters] OF UDT_JC_DepIdleSlotSetType;
  g_transporter   : ARRAY[1..MAX_Transporters] OF UDT_TransporterStatusType;
END_VAR
VAR
  qi       : INT;      (* queue index *)
  si       : INT;      (* slot index *)
  cnt      : INT;      (* task count for this transporter *)
  prev_end : LINT;     (* end time of previous task *)
  prev_sink : INT;     (* sink station of previous task *)
  gap_start : LINT;
  gap_end   : LINT;
  HORIZON  : LINT := 9999999999;   (* open-ended future — must exceed max unix timestamp *)
END_VAR

(* Guard *)
IF i_trans < 1 OR i_trans > MAX_Transporters THEN
  RETURN;
END_IF;

(* Reset output *)
g_dep_idle_slot[i_trans].Count := 0;
si := 0;
cnt := g_task[i_trans].Count;

prev_end  := i_time_s;
(* G05: Use transporter's current station as first-slot anchor *)
prev_sink := g_transporter[i_trans].CurrentStation;

FOR qi := 1 TO MAX_Units DO
  IF qi > cnt THEN
    EXIT;
  END_IF;

  gap_start := prev_end;
  gap_end   := g_task[i_trans].Queue[qi].StartTime;

  (* Only create slot if there is a meaningful gap *)
  IF gap_end > gap_start + LINT#1 THEN
    si := si + 1;
    IF si <= DEP_MAX_IDLE_SLOTS THEN
      g_dep_idle_slot[i_trans].Slots[si].StartTime   := gap_start;
      g_dep_idle_slot[i_trans].Slots[si].EndTime     := gap_end;
      g_dep_idle_slot[i_trans].Slots[si].LiftStationTarget := prev_sink;
      g_dep_idle_slot[i_trans].Slots[si].SinkStationTarget := g_task[i_trans].Queue[qi].LiftStationTarget;
    END_IF;
  END_IF;

  prev_end  := g_task[i_trans].Queue[qi].FinishTime;
  prev_sink := g_task[i_trans].Queue[qi].SinkStationTarget;
END_FOR;

(* Final slot: after last task → open-ended *)
si := si + 1;
IF si <= DEP_MAX_IDLE_SLOTS THEN
  g_dep_idle_slot[i_trans].Slots[si].StartTime   := prev_end;
  g_dep_idle_slot[i_trans].Slots[si].EndTime     := HORIZON;
  g_dep_idle_slot[i_trans].Slots[si].LiftStationTarget := prev_sink;
  g_dep_idle_slot[i_trans].Slots[si].SinkStationTarget := 0;
END_IF;

g_dep_idle_slot[i_trans].Count := si;

END_FUNCTION_BLOCK

(* ---- DEP_FB_CalcOverlap.st ---- *)
(* ============================================================
   DEP_FB_CalcOverlap — Overlap station detection
   ============================================================
   Identifies stations where multiple transporters can operate
   (task_area ranges overlap).  A station is marked as overlap
   if two or more different transporters have task_area ranges
   that cover it (either lift or sink range).

   Source: departureScheduler.js computeOverlapStations()

   Used by: DEP_FB_Scheduler (CALC phase)
   ============================================================ *)

FUNCTION_BLOCK DEP_FB_CalcOverlap
VAR_EXTERNAL CONSTANT
    MAX_Transporters    : INT;
    MIN_StationIndex : INT;
    MAX_StationIndex   : INT;
END_VAR

VAR_EXTERNAL
  g_cfg         : ARRAY[1..MAX_Transporters] OF UDT_TransporterType;
  g_dep_overlap : UDT_JC_DepOverlapType;
END_VAR
VAR
  station_idx         : INT;
  ti          : INT;
  ai          : INT;
  cover_count : INT;
  covered     : BOOL;
  area        : UDT_TaskArea;
END_VAR

g_dep_overlap.Count := 0;

(* G09: Clear full 0..200 domain first *)
FOR station_idx := 0 TO 200 DO
  g_dep_overlap.Flags[station_idx] := FALSE;
END_FOR;

FOR station_idx := MIN_StationIndex TO MAX_StationIndex DO
  cover_count := 0;

  FOR ti := 1 TO MAX_Transporters DO
    covered := FALSE;
    FOR ai := 1 TO 4 DO
      IF NOT covered THEN
        area := g_cfg[ti].TaskArea[ai];
        (* Station is covered if within lift OR sink range *)
        IF (area.MinLift > 0 AND station_idx >= area.MinLift AND station_idx <= area.MaxLift)
           OR (area.MinSink > 0 AND station_idx >= area.MinSink AND station_idx <= area.MaxSink) THEN
          covered := TRUE;
        END_IF;
      END_IF;
    END_FOR;
    IF covered THEN
      cover_count := cover_count + 1;
    END_IF;
  END_FOR;

  IF cover_count >= 2 THEN
    g_dep_overlap.Flags[station_idx] := TRUE;
    g_dep_overlap.Count := g_dep_overlap.Count + 1;
  ELSE
    g_dep_overlap.Flags[station_idx] := FALSE;
  END_IF;
END_FOR;

END_FUNCTION_BLOCK

(* ---- DEP_FB_FitTaskToSlot.st ---- *)
(* ============================================================
   DEP_FB_FitTaskToSlot — Fit a departure task into idle slots
   ============================================================
   Tries to fit a single waiting-batch task into the idle slots
   of its assigned transporter.  Calculates travel times from
   the previous task's sink to this task's lift, and from this
   task's sink to the next task's lift.

   Source: transporterTaskScheduler.js fitSingleTaskToIdleSlots()

   Flex constraint: delay cannot exceed flex_up × flexUpFactor.
   If no slot fits, o_need_extra_s reports the shortfall for
   backward chaining.

   Used by: DEP_FB_Scheduler (CHECK_ANALYZE phase)
   ============================================================ *)

FUNCTION_BLOCK DEP_FB_FitTaskToSlot
VAR_INPUT
  i_lift_stn     : INT;     (* task lift station *)
  i_sink_stn     : INT;     (* task sink station *)
  i_trans_id     : INT;     (* transporter for this task *)
  i_task_start   : LINT;    (* scheduled task start time (s), unix seconds *)
  i_task_end     : LINT;    (* scheduled task end time (s), unix seconds *)
  i_shift_s      : REAL;    (* pre-applied shift (overlap delay) *)
  i_calc_time_s  : DINT;    (* treatment calc_time (s) *)
  i_max_time_s   : DINT;    (* treatment max_time (s) *)
  i_flex_factor  : REAL;    (* flex_up usage factor, e.g. 0.5 *)
  i_margin_s     : REAL;    (* delay significance threshold (s) *)
  i_conflict_margin_s : REAL; (* slot boundary margin (s), typ. 1.0 *)
END_VAR
VAR_OUTPUT
  o_result : UDT_JC_DepFitResultType;
END_VAR
VAR_EXTERNAL CONSTANT
    MAX_Transporters   : INT;
    DEP_MAX_IDLE_SLOTS : INT;
END_VAR

VAR_EXTERNAL
  g_dep_idle_slot : ARRAY[1..MAX_Transporters] OF UDT_JC_DepIdleSlotSetType;
  g_move          : ARRAY[1..MAX_Transporters] OF UDT_JC_MoveTimesType;
END_VAR
VAR
  si          : INT;
  slot_cnt    : INT;
  slot_start  : LINT;
  slot_end    : LINT;
  from_stn    : INT;    (* previous task's sink or transporter home *)
  to_stn      : INT;    (* next task's lift *)
  travel_to   : REAL;   (* travel time: prev_sink → this lift *)
  travel_from : REAL;   (* travel time: this sink → next_lift *)
  earliest    : LINT;
  latest      : LINT;
  task_dur    : LINT;
  delay       : REAL;
  flex_up     : REAL;
  capped_flex : REAL;
  best_delay  : REAL;
  best_slot   : INT;
  found       : BOOL;
  overflow_best_delay : REAL;   (* best delay among flex-overflow slots *)
  overflow_best_slot  : INT;
  tmp_move    : UDT_JC_MoveTimesType;  (* MATIEC cannot index arrays in FUNCTION args *)
END_VAR

(* Initialize output *)
o_result.Fits         := FALSE;
o_result.DelayTime      := 0;
o_result.NeedExtraTime := 0;
o_result.TaskEndTime   := 0;
o_result.SlotIdx     := 0;
o_result.TransporterId     := i_trans_id;

IF i_trans_id < 1 OR i_trans_id > MAX_Transporters THEN
  RETURN;
END_IF;

task_dur   := i_task_end - i_task_start;
flex_up    := DINT_TO_REAL(i_max_time_s - i_calc_time_s);
IF flex_up < 0.0 THEN flex_up := 0.0; END_IF;
capped_flex := flex_up * i_flex_factor;

slot_cnt   := g_dep_idle_slot[i_trans_id].Count;
best_delay := 1.0E9;
best_slot  := 0;
found      := FALSE;
overflow_best_delay := 1.0E9;
overflow_best_slot  := 0;

tmp_move := g_move[i_trans_id];
FOR si := 1 TO DEP_MAX_IDLE_SLOTS DO
  IF si > slot_cnt THEN
    EXIT;
  END_IF;

  slot_start := g_dep_idle_slot[i_trans_id].Slots[si].StartTime;
  slot_end   := g_dep_idle_slot[i_trans_id].Slots[si].EndTime;

  (* ── Travel time: prev task sink → this lift ── *)
  from_stn := g_dep_idle_slot[i_trans_id].Slots[si].LiftStationTarget;
  travel_to := 0.0;
  IF from_stn > 0 AND from_stn <> i_lift_stn THEN
    travel_to := STC_CalcHorizontalTravel(i_from_stn := from_stn, i_to_stn := i_lift_stn, i_move := tmp_move);
  END_IF;

  (* ── Travel time: this sink → next task lift ── *)
  to_stn := g_dep_idle_slot[i_trans_id].Slots[si].SinkStationTarget;
  travel_from := 0.0;
  IF to_stn > 0 AND to_stn <> i_sink_stn THEN
    travel_from := STC_CalcHorizontalTravel(i_from_stn := i_sink_stn, i_to_stn := to_stn, i_move := tmp_move);
  END_IF;

  (* Earliest start = max(slot_start, task_start + shift) + travel_to + conflict_margin *)
  IF slot_start > (i_task_start + REAL_TO_LINT(i_shift_s)) THEN
    earliest := slot_start + REAL_TO_LINT(travel_to + i_conflict_margin_s);
  ELSE
    earliest := i_task_start + REAL_TO_LINT(i_shift_s + travel_to + i_conflict_margin_s);
  END_IF;

  (* Latest end = slot_end - travel_from - conflict_margin *)
  IF slot_end > LINT#9000000000 THEN
    (* Open-ended slot *)
    latest := LINT#9000000000;
  ELSE
    latest := slot_end - REAL_TO_LINT(travel_from + i_conflict_margin_s);
  END_IF;

  (* Check if task fits *)
  IF earliest + task_dur <= latest THEN
    delay := LINT_TO_REAL(earliest - i_task_start) - i_shift_s;
    IF delay < 0.0 THEN delay := 0.0; END_IF;

    (* Flex constraint: small delays always OK; larger must be within flex + 1s *)
    IF delay <= i_margin_s OR delay <= capped_flex + 1.0 THEN
      IF delay < best_delay THEN
        best_delay := delay;
        best_slot  := si;
        found      := TRUE;
      END_IF;
    ELSE
      (* Flex overflow — track separately for backward chaining *)
      IF delay < overflow_best_delay THEN
        overflow_best_delay := delay;
        overflow_best_slot  := si;
      END_IF;
    END_IF;
  END_IF;
END_FOR;

IF found THEN
  o_result.Fits      := TRUE;
  o_result.DelayTime   := REAL_TO_DINT(best_delay);
  o_result.SlotIdx  := best_slot;
  o_result.TaskEndTime := i_task_start + REAL_TO_LINT(i_shift_s + best_delay) + task_dur;
  o_result.NeedExtraTime := 0;
ELSE
  (* Report how much extra is needed for backward chaining *)
  o_result.Fits := FALSE;
  IF overflow_best_delay < 1.0E8 THEN
    (* Overflow slot found — report shortfall beyond capped flex *)
    o_result.DelayTime      := REAL_TO_DINT(overflow_best_delay);
    o_result.NeedExtraTime := REAL_TO_DINT(overflow_best_delay - capped_flex);
    IF o_result.NeedExtraTime < 0 THEN
      o_result.NeedExtraTime := 0;
    END_IF;
  ELSE
    (* No slot at all *)
    o_result.NeedExtraTime := 0;
  END_IF;
END_IF;

END_FUNCTION_BLOCK

(* ---- DEP_FB_OverlapDelay.st ---- *)
(* ============================================================
   DEP_FB_OverlapDelay — Overlap conflict delay calculation
   ============================================================
   When a new task uses a station in the overlap zone (covered
   by multiple transporters), checks for time conflicts with
   tasks on OTHER transporters at the same station.

   Iteratively calculates the minimum delay needed to avoid
   overlap conflicts (max 20 iterations).

   Source: departureScheduler.js calculateOverlapDelay()

   Used by: DEP_FB_Scheduler / DEP_FB_FitTaskToSlot
   ============================================================ *)

FUNCTION_BLOCK DEP_FB_OverlapDelay
VAR_INPUT
  i_lift_stn   : INT;     (* task lift station *)
  i_sink_stn   : INT;     (* task sink station *)
  i_trans_id   : INT;     (* task transporter id *)
  i_task_start : LINT;    (* task start time (s), already shifted *)
  i_task_end   : LINT;    (* task end time (s), already shifted *)
  i_margin_s   : REAL;    (* conflict margin (s), default 1.0 *)
END_VAR
VAR_OUTPUT
  o_delay_s : REAL;       (* total delay needed (s), 0 = no conflict *)
END_VAR
VAR_EXTERNAL CONSTANT
    MAX_Transporters    : INT;
    MIN_StationIndex : INT;
    MAX_StationIndex   : INT;
    MAX_Units           : INT;
    DEP_MAX_DELAY_ACTS  : INT;
END_VAR

VAR_EXTERNAL
  g_task       : ARRAY[1..MAX_Transporters] OF UDT_JC_TskQueueType;
  g_dep_overlap : UDT_JC_DepOverlapType;
END_VAR
VAR
  lift_is_overlap : BOOL;
  sink_is_overlap : BOOL;
  round    : INT;
  ti       : INT;    (* transporter index *)
  qi       : INT;    (* queue index *)
  max_conf : REAL;   (* maximum conflict in this round *)
  t_start  : LINT;   (* shifted task start *)
  t_end    : LINT;   (* shifted task end *)
  e_start  : LINT;   (* existing task start *)
  e_end    : LINT;   (* existing task end *)
  e_lift   : INT;
  e_sink   : INT;
  has_ovlp : BOOL;
  needed   : REAL;
END_VAR

o_delay_s := 0.0;

(* Check if lift/sink are in overlap zone — G09: domain 0..200 *)
IF i_lift_stn >= 0 AND i_lift_stn <= 200 THEN
  lift_is_overlap := g_dep_overlap.Flags[i_lift_stn];
ELSE
  lift_is_overlap := FALSE;
END_IF;
IF i_sink_stn >= 0 AND i_sink_stn <= 200 THEN
  sink_is_overlap := g_dep_overlap.Flags[i_sink_stn];
ELSE
  sink_is_overlap := FALSE;
END_IF;

(* No overlap stations involved → no delay *)
IF NOT lift_is_overlap AND NOT sink_is_overlap THEN
  RETURN;
END_IF;

(* Iterative conflict resolution — max DEP_MAX_DELAY_ACTS rounds *)
FOR round := 1 TO DEP_MAX_DELAY_ACTS DO
  max_conf := 0.0;
  t_start  := i_task_start + REAL_TO_LINT(o_delay_s);
  t_end    := i_task_end + REAL_TO_LINT(o_delay_s);

  (* Check all tasks on OTHER transporters *)
  FOR ti := 1 TO MAX_Transporters DO
    IF ti <> i_trans_id THEN
      FOR qi := 1 TO MAX_Units DO
        IF qi > g_task[ti].Count THEN
          EXIT;
        END_IF;

        e_lift  := g_task[ti].Queue[qi].LiftStationTarget;
        e_sink  := g_task[ti].Queue[qi].SinkStationTarget;
        e_start := g_task[ti].Queue[qi].StartTime;
        e_end   := g_task[ti].Queue[qi].FinishTime;

        (* ★ G08: Zone membership — does existing task use ANY overlap station? *)
        has_ovlp := FALSE;
        IF e_lift >= 0 AND e_lift <= 200 THEN
          IF g_dep_overlap.Flags[e_lift] THEN
            has_ovlp := TRUE;
          END_IF;
        END_IF;
        IF NOT has_ovlp AND e_sink >= 0 AND e_sink <= 200 THEN
          IF g_dep_overlap.Flags[e_sink] THEN
            has_ovlp := TRUE;
          END_IF;
        END_IF;

        IF has_ovlp THEN
          (* Time overlap check: task overlaps with existing? *)
          IF t_start < (e_end + REAL_TO_LINT(i_margin_s)) AND t_end > (e_start - REAL_TO_LINT(i_margin_s)) THEN
            needed := LINT_TO_REAL(e_end - t_start) + i_margin_s;
            IF needed > max_conf THEN
              max_conf := needed;
            END_IF;
          END_IF;
        END_IF;

      END_FOR;  (* qi *)
    END_IF;
  END_FOR;  (* ti *)

  (* No conflict found → done *)
  IF max_conf <= 0.0 THEN
    EXIT;
  END_IF;
  o_delay_s := o_delay_s + max_conf;
END_FOR;  (* round *)

END_FUNCTION_BLOCK

(* ---- DEP_FB_Sandbox.st ---- *)
(* ============================================================
   DEP_FB_Sandbox — Sandbox snapshot / restore / clear
   ============================================================
   Copies global scheduler state to/from the departure sandbox.
   Struct assignment `a := b` in ST copies all fields automatically.

   Source: departureScheduler.js _copyDepartureSandbox()

   Commands:
     1 = SNAPSHOT  — copy globals → g_dep_sandbox
     2 = RESTORE   — copy g_dep_sandbox → globals
     3 = CLEAR     — invalidate sandbox

   Used by: DEP_FB_Scheduler (INIT, REJECT, ACTIVATE)
   ============================================================ *)

FUNCTION_BLOCK DEP_FB_Sandbox
VAR_INPUT
  i_cmd : INT;     (* 1=SNAPSHOT, 2=RESTORE, 3=CLEAR *)
END_VAR
VAR_EXTERNAL CONSTANT
    MAX_Transporters : INT;
    MAX_Units        : INT;
END_VAR

VAR_EXTERNAL
  g_schedule    : ARRAY[1..MAX_Units] OF UDT_JC_TskScheduleType;
  g_batch     : ARRAY[1..MAX_Units] OF UDT_BatchType;
  g_program    : ARRAY[1..MAX_Units] OF UDT_TreatmentProgramType;
  g_task       : ARRAY[1..MAX_Transporters] OF UDT_JC_TskQueueType;
  g_dep_sandbox : UDT_JC_DepSandboxType;
END_VAR
VAR
  ui : INT;
  ti : INT;
END_VAR

IF i_cmd = 1 THEN
  (* ── SNAPSHOT: globals → sandbox ── *)
  FOR ui := 1 TO MAX_Units DO
    g_dep_sandbox.Schedule[ui] := g_schedule[ui];
    g_dep_sandbox.Batches[ui]  := g_batch[ui];
    g_dep_sandbox.Programs[ui] := g_program[ui];
  END_FOR;
  FOR ti := 1 TO MAX_Transporters DO
    g_dep_sandbox.Tasks[ti] := g_task[ti];
  END_FOR;
  g_dep_sandbox.Valid := TRUE;

ELSIF i_cmd = 2 THEN
  (* ── RESTORE: sandbox → globals ── *)
  (* Only restore entries that existed at snapshot time.
     Gateway may have loaded new programs/batches between
     snapshot and restore — protect those writes. *)
  IF g_dep_sandbox.Valid THEN
    FOR ui := 1 TO MAX_Units DO
      g_schedule[ui] := g_dep_sandbox.Schedule[ui];
      IF g_dep_sandbox.Batches[ui].BatchCode > 0 THEN
        g_batch[ui]  := g_dep_sandbox.Batches[ui];
      END_IF;
      IF g_dep_sandbox.Programs[ui].ProgramId > 0 THEN
        g_program[ui] := g_dep_sandbox.Programs[ui];
      END_IF;
    END_FOR;
    FOR ti := 1 TO MAX_Transporters DO
      g_task[ti] := g_dep_sandbox.Tasks[ti];
    END_FOR;
  END_IF;

ELSIF i_cmd = 3 THEN
  (* ── CLEAR: invalidate sandbox ── *)
  g_dep_sandbox.Valid := FALSE;

END_IF;

END_FUNCTION_BLOCK
